PROGRAM MAIN
VAR
END_VAR

//Hallo

END_PROGRAM

(* stored: Version 1.1.0.1, ProductVersion 3.1.4024.9
   POU MAIN: Id {ed26b861-e3c6-47aa-afd8-ee2b6b5c557d}, SpecialFunc None *)
